INTERFACE INTERNAL _I_Thread EXTENDS I_Debug, I_ValidateInterface

METHOD INTERNAL AttachExecute : Result
VAR_INPUT
	iExecute: _I_Execute;
END_VAR
END_METHOD

METHOD INTERNAL AttachWorker : Result
VAR_INPUT
	iWorker: I_Worker;
END_VAR
END_METHOD

METHOD INTERNAL DetachExecute : Result
VAR_INPUT
	iExecute: _I_Execute;
END_VAR
END_METHOD

METHOD INTERNAL DetachWorker : Result
VAR_INPUT
	iWorker: I_Worker;
END_VAR
END_METHOD

END_INTERFACE

(* stored: Version 1.1.0.1
   Itf _I_Thread: Id {a9568707-b22e-4555-9884-6d4e1026cc8c}
   Method AttachExecute: Id {0535368c-1e65-495c-bfb4-5ad515b03a41}
   Method AttachWorker: Id {7f94a2a0-c190-4191-8748-c53f74504f85}
   Method DetachExecute: Id {6c975bb5-71be-43a0-a457-e4cc7c2e9c68}
   Method DetachWorker: Id {8e8574ae-ed06-4a80-9809-8071cc0a41bb} *)
